PROGRAM POWER
VAR
	MC_Power_1: MC_Power;
	MC_Power_2: MC_Power;
	MC_Power_3: MC_Power;
	MC_Power_4: MC_Power;
	MC_Power_5: MC_Power;
	MC_Power_6: MC_Power;
	
END_VAR

MC_Power_1(
	Axis:= AXIS.Axis1, 
	Enable:= POWER_Enable1, 
	Enable_Positive:= POWER_Enable1, 
	Enable_Negative:= POWER_Enable1, 
	Override:= , 
	BufferMode:= , 
	Options:= , 
	Status=> MC_Power_Outputs1.Done, 
	Busy=> MC_Power_Outputs1.Busy, 
	Active=> MC_Power_Outputs1.Active, 
	Error=> MC_Power_Outputs1.Error, 
	ErrorID=> MC_Power_Outputs1.ErrorID);
	
MC_Power_2(
	Axis:= AXIS.Axis2, 
	Enable:= POWER_Enable2, 
	Enable_Positive:= POWER_Enable2, 
	Enable_Negative:= POWER_Enable2, 
	Override:= , 
	BufferMode:= , 
	Options:= , 
	Status=> MC_Power_Outputs2.Done, 
	Busy=> MC_Power_Outputs2.Busy, 
	Active=> MC_Power_Outputs2.Active, 
	Error=> MC_Power_Outputs2.Error, 
	ErrorID=> MC_Power_Outputs2.ErrorID);
	
MC_Power_3(
	Axis:= AXIS.Axis3, 
	Enable:= POWER_Enable3, 
	Enable_Positive:= POWER_Enable3, 
	Enable_Negative:= POWER_Enable3, 
	Override:= , 
	BufferMode:= , 
	Options:= , 
	Status=> MC_Power_Outputs3.Done, 
	Busy=> MC_Power_Outputs3.Busy, 
	Active=> MC_Power_Outputs3.Active, 
	Error=> MC_Power_Outputs3.Error, 
	ErrorID=> MC_Power_Outputs3.ErrorID);
	
MC_Power_4(
	Axis:= AXIS.Axis4, 
	Enable:= POWER_Enable4, 
	Enable_Positive:= POWER_Enable4, 
	Enable_Negative:= POWER_Enable4, 
	Override:= , 
	BufferMode:= , 
	Options:= , 
	Status=> MC_Power_Outputs4.Done, 
	Busy=> MC_Power_Outputs4.Busy, 
	Active=> MC_Power_Outputs4.Active, 
	Error=> MC_Power_Outputs4.Error, 
	ErrorID=> MC_Power_Outputs4.ErrorID);
	
MC_Power_5(
	Axis:= AXIS.Axis5, 
	Enable:= POWER_Enable5, 
	Enable_Positive:= POWER_Enable5, 
	Enable_Negative:= POWER_Enable5, 
	Override:= , 
	BufferMode:= , 
	Options:= , 
	Status=> MC_Power_Outputs5.Done, 
	Busy=> MC_Power_Outputs5.Busy, 
	Active=> MC_Power_Outputs5.Active, 
	Error=> MC_Power_Outputs5.Error, 
	ErrorID=> MC_Power_Outputs5.ErrorID);
	
MC_Power_6(
	Axis:= AXIS.Axis6, 
	Enable:= POWER_Enable6, 
	Enable_Positive:= POWER_Enable6, 
	Enable_Negative:= POWER_Enable6, 
	Override:= , 
	BufferMode:= , 
	Options:= , 
	Status=> MC_Power_Outputs6.Done, 
	Busy=> MC_Power_Outputs6.Busy, 
	Active=> MC_Power_Outputs6.Active, 
	Error=> MC_Power_Outputs6.Error, 
	ErrorID=> MC_Power_Outputs6.ErrorID);

END_PROGRAM

(* stored: Version 1.1.0.1, ProductVersion 3.1.4024.0
   POU POWER: Id {27c3957e-14bf-43e2-90dd-82d4ecc4ca1c}, SpecialFunc None *)
